TYPE ST_M3SelectorIO EXTENDS ST_M2SelectorIO:
STRUCT
	
	i_mfmFlow		AT	%I*	:	REAL;
	i_RawUnit		AT %I*	:	UDINT;
	
END_STRUCT
END_TYPE

(* stored: Version 1.1.0.1, ProductVersion 3.1.4020.12
   DUT ST_M3SelectorIO: Id {312b2dba-2603-45b3-923b-4fd923e08057} *)
